   VAR_IN_OUT
      iqUDT_FifoRcvHeader : "UDT_FifoHeader";   // FIFO receive header
      iqs_FifoRcvData : Array[*] of "UDT_Message";   // FIFO receive data
      iqUDT_FifoMedPriorityHLC : "UDT_FifoHeader";   // FIFO UDS send Header
      iqa_FifoMedPriorityHLC : Array[*] of "UDT_Message";   // FIFO UDS send data
      iqUDT_HLCCommands : "UDT_FedExCommands";   // Commands from UDS
      iqUDT_DA : Struct   // Destination assignment message
         NewMessage : Bool;   // New message received from UDS
         Data : "UDT_FedExMessageDaRa";   // Destination assignment message body
      END_STRUCT;
      iqUDT_RA : Struct   // Destination re-assignment message
         NewMessage : Bool;   // New message received from UDS
         Data : "UDT_FedExMessageDaRa";   // Destination re-assignment message body
      END_STRUCT;
      iqUDT_CD : Struct   // Command message
         NewMessage : Bool;   // New message received from UDS
         Data : "UDT_FedExMessageCD";   // Command message body
      END_STRUCT;
      iqUDT_PS : Struct   // Parameters set message
         NewMessage : Bool;   // New message received from UDS
         Data : "UDT_FedExMessagePS";   // Parameters set message body
      END_STRUCT;
      iqUDT_CustomerIDReference : "UDT_FedExCustomerID";
      iqx_SendHB { ExternalAccessible := 'False'; ExternalVisible := 'False'; ExternalWritable := 'False'} : Bool;   // Send heartbeat request
      iqx_ResetListeningTimer { ExternalAccessible := 'False'; ExternalVisible := 'False'; ExternalWritable := 'False'} : Bool;   // Reset listening time in Heartbeat block
      iq_LoginOK { ExternalAccessible := 'False'; ExternalVisible := 'False'; ExternalWritable := 'False'} : Bool;   // Login in UDS ok
   END_VAR

   VAR
      sFB_FedExLoginResponse { ExternalAccessible := 'False'; ExternalVisible := 'False'; ExternalWritable := 'False'; S7_SetPoint := 'False'} : "FB_FedExLoginResponse";   // Login request send
      sUDT_Facillity { ExternalAccessible := 'False'; ExternalVisible := 'False'; ExternalWritable := 'False'; S7_SetPoint := 'False'} : "UDT_FedExFacility";   // System configuration
      sUDT_MSGHeader { ExternalAccessible := 'False'; ExternalVisible := 'False'; ExternalWritable := 'False'; S7_SetPoint := 'False'} : "UDT_FedExMessageHeader";   // Message header
      sUDT_FifoMsg { ExternalAccessible := 'False'; ExternalVisible := 'False'; ExternalWritable := 'False'; S7_SetPoint := 'False'} : "UDT_Message";   // Buffer for fifos message
      sa_Status { ExternalAccessible := 'False'; ExternalVisible := 'False'; ExternalWritable := 'False'} : Struct   // Status structure
         FIFORcvStatus { ExternalAccessible := 'False'; ExternalVisible := 'False'; ExternalWritable := 'False'} : "UDT_FifoStatus";   // Receive FIFO status structure
         FIFOError { ExternalAccessible := 'False'; ExternalVisible := 'False'; ExternalWritable := 'False'; S7_SetPoint := 'True'} : Bool;   // FIFO error
         FIFOWarning { ExternalAccessible := 'False'; ExternalVisible := 'False'; ExternalWritable := 'False'; S7_SetPoint := 'True'} : Bool;   // FIFO warning
         InvalidCommandCode { ExternalAccessible := 'False'; ExternalVisible := 'False'; ExternalWritable := 'False'} : Bool;   // Invalid command code
         InvalidType { ExternalAccessible := 'False'; ExternalVisible := 'False'; ExternalWritable := 'False'; S7_SetPoint := 'True'} : Bool;   // Invalid message type
         InvalidParameterID { ExternalAccessible := 'False'; ExternalVisible := 'False'; ExternalWritable := 'False'} : Bool;   // Invalig parameter ID
         InvalidLength { ExternalAccessible := 'False'; ExternalVisible := 'False'; ExternalWritable := 'False'} : Bool;   // Received message length is different than programmed
      END_STRUCT;
      st_TimeToSet {InstructionName := 'DTL'; LibVersion := '1.0'; ExternalAccessible := 'False'; ExternalVisible := 'False'; ExternalWritable := 'False'} : DTL;   // Time received from HLC used to set time in the PLC
      ss_NNNNNN { ExternalAccessible := 'False'; ExternalVisible := 'False'; ExternalWritable := 'False'} : String[6];   // GIN number extracted from Package ID
      ss_SS { ExternalAccessible := 'False'; ExternalVisible := 'False'; ExternalWritable := 'False'} : String[2];   // Maximum frequency of the messages
      ss_SorterNumber { ExternalAccessible := 'False'; ExternalVisible := 'False'; ExternalWritable := 'False'} : String;   // Sorter number
      ss_DiverterNumber { ExternalAccessible := 'False'; ExternalVisible := 'False'; ExternalWritable := 'False'} : String;   // Diverter number
      si_GIN { ExternalAccessible := 'False'; ExternalVisible := 'False'; ExternalWritable := 'False'} : Int;   // Gin number converted from string to int
      si_ChuteNumber { ExternalAccessible := 'False'; ExternalVisible := 'False'; ExternalWritable := 'False'} : Int;   // Chute number to enable/disable purge
      si_SS { ExternalAccessible := 'False'; ExternalVisible := 'False'; ExternalWritable := 'False'} : Int;   // Maximum frequency of the messages
      si_i { ExternalAccessible := 'False'; ExternalVisible := 'False'; ExternalWritable := 'False'} : Int;   // Loop counter
      si_PositionOfSpace { ExternalAccessible := 'False'; ExternalVisible := 'False'; ExternalWritable := 'False'} : Int;   // Position of spaces used to remove spaces
      si_MessageLegth { ExternalAccessible := 'False'; ExternalVisible := 'False'; ExternalWritable := 'False'} : Int;   // Received message length
      si_ComValueLen { ExternalAccessible := 'False'; ExternalVisible := 'False'; ExternalWritable := 'False'} : Int;   // Command value length
      si_SpacePositionComValue { ExternalAccessible := 'False'; ExternalVisible := 'False'; ExternalWritable := 'False'} : Int;   // Position of spaces used to remove spaces
      si_WriteTimeStatus { ExternalAccessible := 'False'; ExternalVisible := 'False'; ExternalWritable := 'False'} : Int;   // WR_LOC_T Status
      si_CustomerID { ExternalAccessible := 'False'; ExternalVisible := 'False'; ExternalWritable := 'False'} : Int;
      sx_FacialityCheck { ExternalAccessible := 'False'; ExternalVisible := 'False'; ExternalWritable := 'False'} : Bool;   // When TRUE received faciality configuration is the same as configured in the PLC
      sx_LogOffRequest { ExternalAccessible := 'False'; ExternalVisible := 'False'; ExternalWritable := 'False'} : Bool;   // Log off request from UDS
   END_VAR

   VAR_TEMP
      tx_MsgRead : Bool;   // Message read from FIFO
   END_VAR

   VAR CONSTANT
      cs_DA : String := 'DA';   // Destination assignment message type
      cs_RA : String := 'RA';   // Destination re-assignment message type
      cs_HB : String := 'HB';   // Heartbeat message type
      cs_LI : String := 'LI';   // Login request message type
      cs_LS : String := 'LS';   // Log-off message type
      cs_CD : String := 'CD';   // Command message type
      cs_PS : String := 'PS';   // Parameter set message type
      ci_SizeDAMessage : Int := 213;   // Destination assignment message length
      ci_SizeRAMessage : Int := 213;   // Destination re-assignment message length
      ci_SizeLIMessage : Int := 35;   // Login request message length
      ci_SizeCDMessage : Int := 113;   // Command message length
      ci_SizePSMessage : Int := 129;   // Parameter set message length
   END_VAR


BEGIN
	(*
	----------------------------------------------------------------------------------------

	Version history:
	Date        | Version   | Author        | Remark
	----------------------------------------------------------------------------------------
	22/07/2021  | 1.0       | J.Krawczuk    | first release MHS TIA 15.1
	11/04/2022  | 1.1       | K.Pokorski    | Review
	21/02/2023  | 4.0       | F.Baten       | 4.0 Release TIA 17.5
	*)

	REGION 1 – FIFO header status update

	    // Mode 'S' - FIFO register status update
	    "FC_Fifo"(ic_Mode := 'S',
	              qUDT_Status => #sa_Status.FIFORcvStatus,
	              qx_Error => #sa_Status.FIFOError,
	              qx_Warning => #sa_Status.FIFOWarning,
	              iqv_Data := #sUDT_FifoMsg,
	              iqUDT_FifoHeader := #iqUDT_FifoRcvHeader,
	              iqv_DataBuffer := #iqs_FifoRcvData);

	    IF (NOT #iqUDT_FifoRcvHeader.Status.Empty                             // FIFO not empty
	        AND NOT #sa_Status.FIFOError)                                      // No FIFO error
	    THEN

	        // Mode 'R' - Read FIFO record
	        "FC_Fifo"(ic_Mode := 'R',
	                  qUDT_Status => #sa_Status.FIFORcvStatus,
	                  qx_Error => #sa_Status.FIFOError,
	                  qx_Warning => #sa_Status.FIFOWarning,
	                  iqv_Data := #sUDT_FifoMsg,
	                  iqUDT_FifoHeader := #iqUDT_FifoRcvHeader,
	                  iqv_DataBuffer := #iqs_FifoRcvData);

	        // Message read bit set and position initialize
	        #tx_MsgRead := TRUE;

	        // FIFO empty or FIFO error occured
	    ELSE

	        #tx_MsgRead := FALSE;

	    END_IF;

	END_REGION

	REGION 2 – Decoding header

	    IF #tx_MsgRead      // New message
	    THEN
	        // Header decode
	        "FC_FedExDecodeHeader"(iUDT_FifoMsg := #sUDT_FifoMsg,
	                               qUDT_MSGHeader => #sUDT_MSGHeader);
	    END_IF;
	END_REGION

	REGION 3 - Decoding body

	    IF #tx_MsgRead                                                              // New message
	    THEN
	        #si_MessageLegth := STRING_TO_INT(#sUDT_MSGHeader.MessageLength);      // Convert message length to integer
	        #sa_Status.InvalidType := FALSE;                                        // Invalid type status initialize

	        // Login request message
	        IF #sUDT_MSGHeader.MessageType = #cs_LI
	        THEN

	            // Received message length validation
	            IF #si_MessageLegth = #ci_SizeLIMessage
	            THEN

	                // Faciality ID
	                Chars_TO_Strg(Chars := #sUDT_FifoMsg.Character,
	                              pChars := 7,
	                              Cnt := 6,
	                              Strg => #sUDT_Facillity.FacilityID);

	                // System ID
	                Chars_TO_Strg(Chars := #sUDT_FifoMsg.Character,
	                              pChars := 13,
	                              Cnt := 15,
	                              Strg => #sUDT_Facillity.SystemID);

	                // Version ID
	                Chars_TO_Strg(Chars := #sUDT_FifoMsg.Character,
	                              pChars := 28,
	                              Cnt := 6,
	                              Strg => #sUDT_Facillity.VersionID);

	                // Maximum message frequency
	                Chars_TO_Strg(Chars := #sUDT_FifoMsg.Character,
	                              pChars := 34,
	                              Cnt := 2,
	                              Strg => #ss_SS);

	                // Maximum message frequency conversion to integer
	                #si_SS := STRING_TO_INT(#ss_SS);

	                // For loop to remove spaces from Version ID
	                FOR #si_i := 1 TO 6 DO

	                    #si_PositionOfSpace := 0;
	                    #si_PositionOfSpace := FIND(IN1 := #sUDT_Facillity.VersionID, IN2 := ' ');

	                    IF #si_PositionOfSpace > 0
	                    THEN
	                        #sUDT_Facillity.VersionID := DELETE(IN := #sUDT_Facillity.VersionID, L := 1, P := #si_PositionOfSpace);

	                    END_IF;

	                END_FOR;

	                // Checking if received facility configuration matches configuration in the PLC
	                #sx_FacialityCheck := #iUDT_FacilitySystem.FacilityID = #sUDT_Facillity.FacilityID
	                AND #iUDT_FacilitySystem.SystemID = #sUDT_Facillity.SystemID
	                AND #iUDT_FacilitySystem.VersionID = #sUDT_Facillity.VersionID
	                AND #iUDT_FacilitySystem.SS = #si_SS;

	                // Login response message send
	                #sFB_FedExLoginResponse(iUDT_Facility := #iUDT_FacilityPLC,
	                                        is_LastHost := #is_LastHost,
	                                        ix_ConnectionStatus := #sx_FacialityCheck,
	                                        iqUDT_FifoHeader := #iqUDT_FifoMedPriorityHLC,
	                                        iqa_FifoData := #iqa_FifoMedPriorityHLC);

	                #iqx_ResetListeningTimer := TRUE;
	                #iq_LoginOK := #sx_FacialityCheck;
	            ELSE

	                // In case when received message length is different than programmed set error
	                #sa_Status.InvalidLength := TRUE;

	            END_IF;

	            // Log-off request message
	        ELSIF #sUDT_MSGHeader.MessageType = #cs_LS
	        THEN
	            #sx_LogOffRequest := TRUE;

	            // Destination assignment message
	        ELSIF #sUDT_MSGHeader.MessageType = #cs_DA
	        THEN

	            // Received message length validation
	            IF #si_MessageLegth = #ci_SizeDAMessage
	            THEN

	                // LLC system ID
	                Chars_TO_Strg(Chars := #sUDT_FifoMsg.Character,
	                              pChars := 7,
	                              Cnt := 15,
	                              Strg => #iqUDT_DA.Data.LLCSystemID);

	                // Package ID
	                Chars_TO_Strg(Chars := #sUDT_FifoMsg.Character,
	                              pChars := 22,
	                              Cnt := 15,
	                              Strg => #iqUDT_DA.Data.PackageID);

	                // High level package ID
	                Chars_TO_Strg(Chars := #sUDT_FifoMsg.Character,
	                              pChars := 37,
	                              Cnt := 10,
	                              Strg => #iqUDT_DA.Data.HLCPackageID);

	                // Cell number
	                Chars_TO_Strg(Chars := #sUDT_FifoMsg.Character,
	                              pChars := 47,
	                              Cnt := 4,
	                              Strg => #iqUDT_DA.Data.CellNumber);

	                // Destination 1
	                Chars_TO_Strg(Chars := #sUDT_FifoMsg.Character,
	                              pChars := 51,
	                              Cnt := 6,
	                              Strg => #iqUDT_DA.Data.Destination1);

	                // Cut off time destination 1
	                Chars_TO_Strg(Chars := #sUDT_FifoMsg.Character,
	                              pChars := 57,
	                              Cnt := 5,
	                              Strg => #iqUDT_DA.Data.CutOffTimeDestination1);

	                // Destination 2
	                Chars_TO_Strg(Chars := #sUDT_FifoMsg.Character,
	                              pChars := 62,
	                              Cnt := 6,
	                              Strg => #iqUDT_DA.Data.Destination2);

	                // Cut off time destination 2
	                Chars_TO_Strg(Chars := #sUDT_FifoMsg.Character,
	                              pChars := 68,
	                              Cnt := 5,
	                              Strg => #iqUDT_DA.Data.CutOffTimeDestination2);

	                // Destination 3
	                Chars_TO_Strg(Chars := #sUDT_FifoMsg.Character,
	                              pChars := 73,
	                              Cnt := 6,
	                              Strg => #iqUDT_DA.Data.Destination3);

	                // Cut off time destination 3
	                Chars_TO_Strg(Chars := #sUDT_FifoMsg.Character,
	                              pChars := 79,
	                              Cnt := 5,
	                              Strg => #iqUDT_DA.Data.CutOffTimeDestination3);

	                // Destination 4
	                Chars_TO_Strg(Chars := #sUDT_FifoMsg.Character,
	                              pChars := 84,
	                              Cnt := 6,
	                              Strg => #iqUDT_DA.Data.Destination4);

	                // Cut off time destination 4
	                Chars_TO_Strg(Chars := #sUDT_FifoMsg.Character,
	                              pChars := 90,
	                              Cnt := 5,
	                              Strg => #iqUDT_DA.Data.CutOffTimeDestination4);

	                // Destination 5
	                Chars_TO_Strg(Chars := #sUDT_FifoMsg.Character,
	                              pChars := 95,
	                              Cnt := 6,
	                              Strg => #iqUDT_DA.Data.Destination5);

	                // Cut off time destination 5
	                Chars_TO_Strg(Chars := #sUDT_FifoMsg.Character,
	                              pChars := 101,
	                              Cnt := 5,
	                              Strg => #iqUDT_DA.Data.CutOffTimeDestination5);

	                // High level data text
	                Chars_TO_Strg(Chars := #sUDT_FifoMsg.Character,
	                              pChars := 106,
	                              Cnt := 20,
	                              Strg => #iqUDT_DA.Data.HLCDataText);

	                // Barcode data
	                Chars_TO_Strg(Chars := #sUDT_FifoMsg.Character,
	                              pChars := 126,
	                              Cnt := 50,
	                              Strg => #iqUDT_DA.Data.Barcodedata);

	                // Result code
	                Chars_TO_Strg(Chars := #sUDT_FifoMsg.Character,
	                              pChars := 176,
	                              Cnt := 16,
	                              Strg => #iqUDT_DA.Data.HLCResultCode);

	                // Timestamp
	                Chars_TO_Strg(Chars := #sUDT_FifoMsg.Character,
	                              pChars := 192,
	                              Cnt := 17,
	                              Strg => #iqUDT_DA.Data.Timestamp);

	                // Time zone designator
	                Chars_TO_Strg(Chars := #sUDT_FifoMsg.Character,
	                              pChars := 209,
	                              Cnt := 5,
	                              Strg => #iqUDT_DA.Data.TimeZoneDesignator);

	                // Convert 'NNNNNN' part in package ID to GIN number and store data in GIN database
	                #ss_NNNNNN := RIGHT(IN := #iqUDT_DA.Data.PackageID, L := 6);
	                STRG_VAL(IN := #ss_NNNNNN,
	                         FORMAT := 16#0,
	                         P := 1,
	                         OUT => #si_CustomerID);

	                IF #si_CustomerID > 1 AND #si_CustomerID < 999999 THEN
	                    #si_GIN := #iqUDT_CustomerIDReference.CustomerIDReference[#si_CustomerID];
	                END_IF;

	                // Write data from destination assignment message to GIN array
	                IF #si_GIN > 0
	                    AND #si_GIN <= 9999
	                THEN

	                    "DB_GIN".GIN[#si_GIN].FedEx.LLCSystemID := #iqUDT_DA.Data.LLCSystemID;
	                    "DB_GIN".GIN[#si_GIN].FedEx.PackageID := #iqUDT_DA.Data.PackageID;
	                    "DB_GIN".GIN[#si_GIN].FedEx.HLCPackageID := #iqUDT_DA.Data.HLCPackageID;
	                    "DB_GIN".GIN[#si_GIN].FedEx.CellNumber := #iqUDT_DA.Data.CellNumber;
	                    "DB_GIN".GIN[#si_GIN].FedEx.Destination1 := #iqUDT_DA.Data.Destination1;
	                    "DB_GIN".GIN[#si_GIN].FedEx.CutOffTimeDestination1 := #iqUDT_DA.Data.CutOffTimeDestination1;
	                    "DB_GIN".GIN[#si_GIN].FedEx.Destination2 := #iqUDT_DA.Data.Destination2;
	                    "DB_GIN".GIN[#si_GIN].FedEx.CutOffTimeDestination2 := #iqUDT_DA.Data.CutOffTimeDestination2;
	                    "DB_GIN".GIN[#si_GIN].FedEx.Destination3 := #iqUDT_DA.Data.Destination3;
	                    "DB_GIN".GIN[#si_GIN].FedEx.CutOffTimeDestination3 := #iqUDT_DA.Data.CutOffTimeDestination3;
	                    "DB_GIN".GIN[#si_GIN].FedEx.Destination4 := #iqUDT_DA.Data.Destination4;
	                    "DB_GIN".GIN[#si_GIN].FedEx.CutOffTimeDestination4 := #iqUDT_DA.Data.CutOffTimeDestination4;
	                    "DB_GIN".GIN[#si_GIN].FedEx.Destination5 := #iqUDT_DA.Data.Destination5;
	                    "DB_GIN".GIN[#si_GIN].FedEx.CutOffTimeDestination5 := #iqUDT_DA.Data.CutOffTimeDestination5;
	                    "DB_GIN".GIN[#si_GIN].FedEx.HLCDataText := #iqUDT_DA.Data.HLCDataText;
	                    "DB_GIN".GIN[#si_GIN].FedEx.Barcodedata := #iqUDT_DA.Data.Barcodedata;
	                    "DB_GIN".GIN[#si_GIN].FedEx.HLCResultCode := #iqUDT_DA.Data.HLCResultCode;
	                    "DB_GIN".GIN[#si_GIN].FedEx.Timestamp := #iqUDT_DA.Data.Timestamp;
	                    "DB_GIN".GIN[#si_GIN].FedEx.TimeZoneDesignator := #iqUDT_DA.Data.TimeZoneDesignator;

	                    "DB_GIN".GIN[#si_GIN].General.Destination[0] := STRING_TO_DINT(#iqUDT_DA.Data.Destination1);
	                    "DB_GIN".GIN[#si_GIN].General.Destination[1] := STRING_TO_DINT(#iqUDT_DA.Data.Destination2);
	                    "DB_GIN".GIN[#si_GIN].General.Destination[2] := STRING_TO_DINT(#iqUDT_DA.Data.Destination3);
	                    "DB_GIN".GIN[#si_GIN].General.Destination[3] := STRING_TO_DINT(#iqUDT_DA.Data.Destination4);
	                    "DB_GIN".GIN[#si_GIN].General.Destination[4] := STRING_TO_DINT(#iqUDT_DA.Data.Destination5);

	                    #iqUDT_DA.NewMessage := TRUE;
	                    #iqx_ResetListeningTimer := TRUE;

	                END_IF;
	            ELSE
	                // In case when received message length is different than programmed set error
	                #sa_Status.InvalidLength := TRUE;

	            END_IF;

	            // Destination re-assignment message
	        ELSIF #sUDT_MSGHeader.MessageType = #cs_RA
	        THEN

	            // Received message length validation
	            IF #si_MessageLegth = #ci_SizeRAMessage
	            THEN

	                // LLC system ID
	                Chars_TO_Strg(Chars := #sUDT_FifoMsg.Character,
	                              pChars := 7,
	                              Cnt := 15,
	                              Strg => #iqUDT_RA.Data.LLCSystemID);

	                // Package ID
	                Chars_TO_Strg(Chars := #sUDT_FifoMsg.Character,
	                              pChars := 22,
	                              Cnt := 15,
	                              Strg => #iqUDT_RA.Data.PackageID);

	                // High level package ID
	                Chars_TO_Strg(Chars := #sUDT_FifoMsg.Character,
	                              pChars := 37,
	                              Cnt := 10,
	                              Strg => #iqUDT_RA.Data.HLCPackageID);

	                // Cell number
	                Chars_TO_Strg(Chars := #sUDT_FifoMsg.Character,
	                              pChars := 47,
	                              Cnt := 4,
	                              Strg => #iqUDT_RA.Data.CellNumber);

	                // Destination 1
	                Chars_TO_Strg(Chars := #sUDT_FifoMsg.Character,
	                              pChars := 51,
	                              Cnt := 6,
	                              Strg => #iqUDT_RA.Data.Destination1);

	                // Cut off time destination 1
	                Chars_TO_Strg(Chars := #sUDT_FifoMsg.Character,
	                              pChars := 57,
	                              Cnt := 5,
	                              Strg => #iqUDT_RA.Data.CutOffTimeDestination1);

	                // Destination 2
	                Chars_TO_Strg(Chars := #sUDT_FifoMsg.Character,
	                              pChars := 62,
	                              Cnt := 6,
	                              Strg => #iqUDT_RA.Data.Destination2);

	                // Cut off time destination 2
	                Chars_TO_Strg(Chars := #sUDT_FifoMsg.Character,
	                              pChars := 68,
	                              Cnt := 5,
	                              Strg => #iqUDT_RA.Data.CutOffTimeDestination2);

	                // Destination 3
	                Chars_TO_Strg(Chars := #sUDT_FifoMsg.Character,
	                              pChars := 73,
	                              Cnt := 6,
	                              Strg => #iqUDT_RA.Data.Destination3);

	                // Cut off time destination 3
	                Chars_TO_Strg(Chars := #sUDT_FifoMsg.Character,
	                              pChars := 79,
	                              Cnt := 5,
	                              Strg => #iqUDT_RA.Data.CutOffTimeDestination3);

	                // Destination 4
	                Chars_TO_Strg(Chars := #sUDT_FifoMsg.Character,
	                              pChars := 84,
	                              Cnt := 6,
	                              Strg => #iqUDT_RA.Data.Destination4);

	                // Cut off time destination 4
	                Chars_TO_Strg(Chars := #sUDT_FifoMsg.Character,
	                              pChars := 90,
	                              Cnt := 5,
	                              Strg => #iqUDT_RA.Data.CutOffTimeDestination4);

	                // Destination 5
	                Chars_TO_Strg(Chars := #sUDT_FifoMsg.Character,
	                              pChars := 95,
	                              Cnt := 6,
	                              Strg => #iqUDT_RA.Data.Destination5);

	                // Cut off time destination 5
	                Chars_TO_Strg(Chars := #sUDT_FifoMsg.Character,
	                              pChars := 101,
	                              Cnt := 5,
	                              Strg => #iqUDT_RA.Data.CutOffTimeDestination5);

	                // High level data text
	                Chars_TO_Strg(Chars := #sUDT_FifoMsg.Character,
	                              pChars := 106,
	                              Cnt := 20,
	                              Strg => #iqUDT_RA.Data.HLCDataText);

	                // Barcode data
	                Chars_TO_Strg(Chars := #sUDT_FifoMsg.Character,
	                              pChars := 126,
	                              Cnt := 50,
	                              Strg => #iqUDT_RA.Data.Barcodedata);

	                // Result code
	                Chars_TO_Strg(Chars := #sUDT_FifoMsg.Character,
	                              pChars := 176,
	                              Cnt := 16,
	                              Strg => #iqUDT_RA.Data.HLCResultCode);

	                // Timestamp
	                Chars_TO_Strg(Chars := #sUDT_FifoMsg.Character,
	                              pChars := 192,
	                              Cnt := 17,
	                              Strg => #iqUDT_RA.Data.Timestamp);

	                // Time zone designator
	                Chars_TO_Strg(Chars := #sUDT_FifoMsg.Character,
	                              pChars := 209,
	                              Cnt := 5,
	                              Strg => #iqUDT_RA.Data.TimeZoneDesignator);

	                // Convert 'NNNNNN' part in package ID to GIN number and store data in GIN database
	                #ss_NNNNNN := RIGHT(IN := #iqUDT_RA.Data.PackageID, L := 6);
	                STRG_VAL(IN := #ss_NNNNNN,
	                         FORMAT := 16#0,
	                         P := 1,
	                         OUT => #si_CustomerID);

	                IF #si_CustomerID > 1 AND #si_CustomerID < 999999 THEN
	                    #si_GIN := #iqUDT_CustomerIDReference.CustomerIDReference[#si_CustomerID];
	                END_IF;

	                // Write data from destination assignment message to GIN array
	                IF #si_GIN > 0
	                    AND #si_GIN <= 9999
	                THEN
	                    "DB_GIN".GIN[#si_GIN].FedEx.LLCSystemID := #iqUDT_RA.Data.LLCSystemID;
	                    "DB_GIN".GIN[#si_GIN].FedEx.PackageID := #iqUDT_RA.Data.PackageID;
	                    "DB_GIN".GIN[#si_GIN].FedEx.HLCPackageID := #iqUDT_RA.Data.HLCPackageID;
	                    "DB_GIN".GIN[#si_GIN].FedEx.CellNumber := #iqUDT_RA.Data.CellNumber;
	                    "DB_GIN".GIN[#si_GIN].FedEx.Destination1 := #iqUDT_RA.Data.Destination1;
	                    "DB_GIN".GIN[#si_GIN].FedEx.CutOffTimeDestination1 := #iqUDT_RA.Data.CutOffTimeDestination1;
	                    "DB_GIN".GIN[#si_GIN].FedEx.Destination2 := #iqUDT_RA.Data.Destination2;
	                    "DB_GIN".GIN[#si_GIN].FedEx.CutOffTimeDestination2 := #iqUDT_RA.Data.CutOffTimeDestination2;
	                    "DB_GIN".GIN[#si_GIN].FedEx.Destination3 := #iqUDT_RA.Data.Destination3;
	                    "DB_GIN".GIN[#si_GIN].FedEx.CutOffTimeDestination3 := #iqUDT_RA.Data.CutOffTimeDestination3;
	                    "DB_GIN".GIN[#si_GIN].FedEx.Destination4 := #iqUDT_RA.Data.Destination4;
	                    "DB_GIN".GIN[#si_GIN].FedEx.CutOffTimeDestination4 := #iqUDT_RA.Data.CutOffTimeDestination4;
	                    "DB_GIN".GIN[#si_GIN].FedEx.Destination5 := #iqUDT_RA.Data.Destination5;
	                    "DB_GIN".GIN[#si_GIN].FedEx.CutOffTimeDestination5 := #iqUDT_RA.Data.CutOffTimeDestination5;
	                    "DB_GIN".GIN[#si_GIN].FedEx.HLCDataText := #iqUDT_RA.Data.HLCDataText;
	                    "DB_GIN".GIN[#si_GIN].FedEx.Barcodedata := #iqUDT_RA.Data.Barcodedata;
	                    "DB_GIN".GIN[#si_GIN].FedEx.HLCResultCode := #iqUDT_RA.Data.HLCResultCode;
	                    "DB_GIN".GIN[#si_GIN].FedEx.Timestamp := #iqUDT_RA.Data.Timestamp;
	                    "DB_GIN".GIN[#si_GIN].FedEx.TimeZoneDesignator := #iqUDT_RA.Data.TimeZoneDesignator;

	                    "DB_GIN".GIN[#si_GIN].General.Destination[0] := STRING_TO_DINT(#iqUDT_RA.Data.Destination1);
	                    "DB_GIN".GIN[#si_GIN].General.Destination[1] := STRING_TO_DINT(#iqUDT_RA.Data.Destination2);
	                    "DB_GIN".GIN[#si_GIN].General.Destination[2] := STRING_TO_DINT(#iqUDT_RA.Data.Destination3);
	                    "DB_GIN".GIN[#si_GIN].General.Destination[3] := STRING_TO_DINT(#iqUDT_RA.Data.Destination4);
	                    "DB_GIN".GIN[#si_GIN].General.Destination[4] := STRING_TO_DINT(#iqUDT_RA.Data.Destination5);

	                    #iqUDT_RA.NewMessage := TRUE;
	                    #iqx_ResetListeningTimer := TRUE;

	                END_IF;

	            ELSE
	                // In case when received message length is different than programmed set error
	                #sa_Status.InvalidLength := TRUE;

	            END_IF;

	            // Command message
	        ELSIF #sUDT_MSGHeader.MessageType = #cs_CD
	        THEN
	            // Received message length validation
	            IF #si_MessageLegth = #ci_SizeCDMessage
	            THEN
	                // Invalid command code initialization
	                #sa_Status.InvalidCommandCode := FALSE;

	                // Command code
	                Chars_TO_Strg(Chars := #sUDT_FifoMsg.Character,
	                              pChars := 7,
	                              Cnt := 3,
	                              Strg => #iqUDT_CD.Data.CommandCode);

	                // Command value
	                Chars_TO_Strg(Chars := #sUDT_FifoMsg.Character,
	                              pChars := 10,
	                              Cnt := 82,
	                              Strg => #iqUDT_CD.Data.CommandValue);

	                // Timestamp
	                Chars_TO_Strg(Chars := #sUDT_FifoMsg.Character,
	                              pChars := 92,
	                              Cnt := 17,
	                              Strg => #iqUDT_CD.Data.Timestamp);

	                // Time zone designator
	                Chars_TO_Strg(Chars := #sUDT_FifoMsg.Character,
	                              pChars := 109,
	                              Cnt := 5,
	                              Strg => #iqUDT_CD.Data.TimeZoneDesignator);

	                #iqUDT_CD.NewMessage := TRUE;
	                #iqx_ResetListeningTimer := TRUE;

	                // Start of sort command
	                IF #iqUDT_CD.Data.CommandCode = '001'
	                THEN
	                    #iqUDT_HLCCommands.StartSort.StartSort := TRUE;
	                    #iqUDT_HLCCommands.EndSort.EndSort := FALSE;
	                    #iqUDT_HLCCommands.StartSort.NewMessage := TRUE;

	                    // End of sort command
	                ELSIF #iqUDT_CD.Data.CommandCode = '002'
	                THEN
	                    #iqUDT_HLCCommands.StartSort.StartSort := FALSE;
	                    #iqUDT_HLCCommands.EndSort.EndSort := TRUE;
	                    #iqUDT_HLCCommands.EndSort.NewMessage := TRUE;
	                    // Upload chute status command
	                ELSIF #iqUDT_CD.Data.CommandCode = '003'
	                THEN
	                    #iqUDT_HLCCommands.UploadChuteStatus.NewMessage := TRUE;

	                    // Upload all equipment status command
	                ELSIF #iqUDT_CD.Data.CommandCode = '004'
	                THEN
	                    #iqUDT_HLCCommands.UploadAllStatus.NewMessage := TRUE;

	                    // Block diverter automated smalls
	                ELSIF #iqUDT_CD.Data.CommandCode = '005'
	                THEN
	                    #ss_SorterNumber := MID(IN := #iqUDT_CD.Data.CommandValue, L := 5, P := 3);
	                    #ss_DiverterNumber := MID(IN := #iqUDT_CD.Data.CommandValue, L := 6, P := 8);
	                    #iqUDT_HLCCommands.BlockDivertSmalls.SorterNumber := (#ss_SorterNumber);
	                    #iqUDT_HLCCommands.BlockDivertSmalls.DivertNumber := (#ss_DiverterNumber);

	                    // Unblock diverter automated smalls
	                ELSIF #iqUDT_CD.Data.CommandCode = '006'
	                THEN

	                    #ss_SorterNumber := MID(IN := #iqUDT_CD.Data.CommandValue, L := 5, P := 3);
	                    #ss_DiverterNumber := MID(IN := #iqUDT_CD.Data.CommandValue, L := 6, P := 8);
	                    #iqUDT_HLCCommands.UnblockDivertSmalls.SorterNumber := (#ss_SorterNumber);
	                    #iqUDT_HLCCommands.UnblockDivertSmalls.DivertNumber := (#ss_DiverterNumber);

	                    // Chute purge enable
	                ELSIF #iqUDT_CD.Data.CommandCode = '007'
	                THEN

	                    // Removing spaces from caommand value
	                    FOR #si_i := 1 TO 82 DO

	                        #si_SpacePositionComValue := FIND(IN1 := #iqUDT_CD.Data.CommandValue, IN2 := ' ');
	                        IF #si_SpacePositionComValue <> 0
	                        THEN
	                            #iqUDT_CD.Data.CommandValue := DELETE(IN := #iqUDT_CD.Data.CommandValue, L := 1, P := #si_SpacePositionComValue);

	                        END_IF;

	                    END_FOR;

	                    #iqUDT_HLCCommands.EnablePurge.PLC := LEFT(IN := #iqUDT_CD.Data.CommandValue, L := 6);
	                    #iqUDT_CD.Data.CommandValue := DELETE(IN := #iqUDT_CD.Data.CommandValue, L := 6, P := 1);
	                    #si_ComValueLen := LEN(#iqUDT_CD.Data.CommandValue);

	                    // Extracting up to 5 chute numbers to enable purge
	                    IF #si_ComValueLen MOD 6 = 0 AND #si_ComValueLen <= 30
	                    THEN

	                        #si_ChuteNumber := 0;

	                        FOR #si_i := (#si_ComValueLen / 6) TO 1 BY -1 DO

	                            #si_ChuteNumber += 1;

	                            #iqUDT_HLCCommands.EnablePurge.Chute[#si_ChuteNumber] := (LEFT(IN := #iqUDT_CD.Data.CommandValue, L := 6));
	                            #iqUDT_CD.Data.CommandValue := DELETE(IN := #iqUDT_CD.Data.CommandValue, L := 6, P := 1);

	                        END_FOR;

	                    END_IF;

	                    // Chute purge disable
	                ELSIF #iqUDT_CD.Data.CommandCode = '008'
	                THEN
	                    // Removing spaces from caommand value
	                    FOR #si_i := 1 TO 82 DO

	                        #si_SpacePositionComValue := FIND(IN1 := #iqUDT_CD.Data.CommandValue, IN2 := ' ');
	                        IF #si_SpacePositionComValue <> 0
	                        THEN
	                            #iqUDT_CD.Data.CommandValue := DELETE(IN := #iqUDT_CD.Data.CommandValue, L := 1, P := #si_SpacePositionComValue);

	                        END_IF;

	                    END_FOR;

	                    #iqUDT_HLCCommands.DisablePurge.PLC := LEFT(IN := #iqUDT_CD.Data.CommandValue, L := 6);
	                    #iqUDT_CD.Data.CommandValue := DELETE(IN := #iqUDT_CD.Data.CommandValue, L := 6, P := 1);
	                    #si_ComValueLen := LEN(#iqUDT_CD.Data.CommandValue);

	                    // Extracting up to 5 chute numbers to disable purge
	                    IF #si_ComValueLen MOD 6 = 0
	                    THEN

	                        #si_ChuteNumber := 0;

	                        FOR #si_i := (#si_ComValueLen / 6) - 1 TO 1 BY -1 DO

	                            #si_ChuteNumber += 1;

	                            #iqUDT_HLCCommands.DisablePurge.Chute[#si_ChuteNumber] := (LEFT(IN := #iqUDT_CD.Data.CommandValue, L := 6));
	                            #iqUDT_CD.Data.CommandValue := DELETE(IN := #iqUDT_CD.Data.CommandValue, L := 6, P := 1);

	                        END_FOR;

	                    END_IF;

	                    // Lamp control
	                ELSIF #iqUDT_CD.Data.CommandCode = '009'
	                THEN

	                    #iqUDT_HLCCommands.ChuteLamp.ChuteNumber := (LEFT(IN := #iqUDT_CD.Data.CommandValue, L := 6));
	                    #iqUDT_HLCCommands.ChuteLamp.Mode := (MID(IN := #iqUDT_CD.Data.CommandValue, L := 1, P := 7));
	                    #iqUDT_HLCCommands.ChuteLamp.Color := (MID(IN := #iqUDT_CD.Data.CommandValue, L := 9, P := 8));

	                ELSE
	                    // In case when received command is different than programmed set error
	                    #sa_Status.InvalidCommandCode := TRUE;

	                END_IF;

	                //    #q_UDT_HLCCommands := #s_UDT_HLCCommands;

	            ELSE
	                // In case when received message length is different than programmed set error
	                #sa_Status.InvalidLength := TRUE;

	            END_IF;

	            // Parameter set message
	        ELSIF #sUDT_MSGHeader.MessageType = #cs_PS
	        THEN

	            // Received message length validation
	            IF #si_MessageLegth = #ci_SizePSMessage
	            THEN

	                // System ID
	                Chars_TO_Strg(Chars := #sUDT_FifoMsg.Character,
	                              pChars := 7,
	                              Cnt := 15,
	                              Strg => #iqUDT_PS.Data.SystemID);

	                // Parameter ID
	                Chars_TO_Strg(Chars := #sUDT_FifoMsg.Character,
	                              pChars := 22,
	                              Cnt := 4,
	                              Strg => #iqUDT_PS.Data.ParameterID);

	                // Parameter value
	                Chars_TO_Strg(Chars := #sUDT_FifoMsg.Character,
	                              pChars := 26,
	                              Cnt := 82,
	                              Strg => #iqUDT_PS.Data.ParameterValue);

	                // Timestamp
	                Chars_TO_Strg(Chars := #sUDT_FifoMsg.Character,
	                              pChars := 108,
	                              Cnt := 17,
	                              Strg => #iqUDT_PS.Data.Timestamp);

	                // Time zone designator
	                Chars_TO_Strg(Chars := #sUDT_FifoMsg.Character,
	                              pChars := 125,
	                              Cnt := 5,
	                              Strg => #iqUDT_PS.Data.TimeZoneDesignator);

	                #iqUDT_PS.NewMessage := TRUE;
	                #iqx_ResetListeningTimer := TRUE;

	                // Set time parameter
	                IF #iqUDT_PS.Data.ParameterID = 'TIME'
	                THEN
	                    // Invalid parameter ID initialization
	                    #sa_Status.InvalidParameterID := FALSE;

	                    // Converting received date and time to DTL format
	                    #st_TimeToSet.YEAR := STRING_TO_UINT(LEFT(IN := #iqUDT_PS.Data.ParameterValue, L := 4));
	                    #st_TimeToSet.MONTH := STRING_TO_USINT(MID(IN := #iqUDT_PS.Data.ParameterValue, L := 2, P := 5));
	                    #st_TimeToSet.DAY := STRING_TO_USINT(MID(IN := #iqUDT_PS.Data.ParameterValue, L := 2, P := 7));
	                    #st_TimeToSet.HOUR := STRING_TO_USINT(MID(IN := #iqUDT_PS.Data.ParameterValue, L := 2, P := 9));
	                    #st_TimeToSet.MINUTE := STRING_TO_USINT(MID(IN := #iqUDT_PS.Data.ParameterValue, L := 2, P := 11));
	                    #st_TimeToSet.SECOND := STRING_TO_USINT(MID(IN := #iqUDT_PS.Data.ParameterValue, L := 2, P := 13));
	                    #st_TimeToSet.NANOSECOND := 0;

	                    // Set time in the PLC
	                    #si_WriteTimeStatus := WR_LOC_T(LOCTIME := #st_TimeToSet, DST := FALSE);

	                ELSE
	                    // In case when received parameter ID is different than programmed set error
	                    #sa_Status.InvalidParameterID := TRUE;

	                END_IF;

	            ELSE
	                // In case when received message length is different than programmed set error
	                #sa_Status.InvalidLength := TRUE;

	            END_IF;

	            // Heartbeat message
	        ELSIF #sUDT_MSGHeader.MessageType = #cs_HB
	        THEN

	            #iqx_SendHB := TRUE;


	        ELSE
	            // In case when received message type is different than programmed set error
	            #sa_Status.InvalidType := TRUE;

	        END_IF;
	    END_IF;

	END_REGION
END_FUNCTION_BLOCK

FUNCTION_BLOCK "FB_FedExDestinationLookupMessage"
TITLE = FB_Heartbeat
{ S7_Optimized_Access := 'TRUE' }
AUTHOR : MHSE
FAMILY : UPS_SpecificCommunication
VERSION : 3.0
// ATTRIBUTES
// AUTO_NUMBER = True
// BLOCK_NUMBER = 67
// END_ATTRIBUTES
//Function block to send and monitor the UPS heartbeat message.
   VAR_INPUT
      iUDT_Facility { ExternalAccessible := 'False'; ExternalVisible := 'False'; ExternalWritable := 'False'} : "UDT_FedExFacility";   // System configuration
      is_LOConEquipment { ExternalAccessible := 'False'; ExternalVisible := 'False'; ExternalWritable := 'False'} : String[3];   // Location of the equipment
      is_DEPCOD { ExternalAccessible := 'False'; ExternalVisible := 'False'; ExternalWritable := 'False'} : String[6];   // Depot Code
      is_TYPofEquipment { ExternalAccessible := 'False'; ExternalVisible := 'False'; ExternalWritable := 'False'} : String[3];   // Type of equipment
      is_NumberOfTheEquipment { ExternalAccessible := 'False'; ExternalVisible := 'False'; ExternalWritable := 'False'} : String[3];   // Number of the equipment 001-999
      is_TrayCellNumber { ExternalAccessible := 'False'; ExternalVisible := 'False'; ExternalWritable := 'False'} : String[3];   // Tray/Cell number (for loop sorters) or generated by LLC (on line sorters).
      is_SorterNumber { ExternalAccessible := 'False'; ExternalVisible := 'False'; ExternalWritable := 'False'} : String[2];   // Sorter number
      is_InductionNumber { ExternalAccessible := 'False'; ExternalVisible := 'False'; ExternalWritable := 'False'} : String[2];   // Induction number
      is_AreaNumber { ExternalAccessible := 'False'; ExternalVisible := 'False'; ExternalWritable := 'False'} : String[2];   // Area number
      ii_Gin { ExternalAccessible := 'False'; ExternalVisible := 'False'; ExternalWritable := 'False'} : Int;   // GIN number
   END_VAR

   VAR_OUTPUT
      qx_Error { ExternalAccessible := 'False'; ExternalVisible := 'False'; ExternalWritable := 'False'} : Bool;   // Error
   END_VAR

   VAR_IN_OUT
      iqUDT_FifoHeader : "UDT_FifoHeader";   // FIFO header
      iqa_FifoData : Array[*] of "UDT_Message";   // FIFO data
      iqx_UnexpectedDLReq { ExternalAccessible := 'False'; ExternalVisible := 'False'; ExternalWritable := 'False'} : Bool;
   END_VAR

   VAR
      sUDT_MessageArray { ExternalAccessible := 'False'; ExternalVisible := 'False'; ExternalWritable := 'False'; S7_SetPoint := 'False'} : "UDT_Message";   // Message character array
      sa_Status { ExternalAccessible := 'False'; ExternalVisible := 'False'; ExternalWritable := 'False'} : Struct   // Status structure
         FIFOStatus { ExternalAccessible := 'False'; ExternalVisible := 'False'; ExternalWritable := 'False'} : "UDT_FifoStatus";   // FIFO status structure
         FIFOError { ExternalAccessible := 'False'; ExternalVisible := 'False'; ExternalWritable := 'False'; S7_SetPoint := 'True'} : Bool;   // FIFO data buffer full
         FIFOWarning { ExternalAccessible := 'False'; ExternalVisible := 'False'; ExternalWritable := 'False'; S7_SetPoint := 'True'} : Bool;   // FIFO error
         InvalidGIN { ExternalAccessible := 'False'; ExternalVisible := 'False'; ExternalWritable := 'False'} : Bool;   //  Invalid GIN
         InvalidMessageLength { ExternalAccessible := 'False'; ExternalVisible := 'False'; ExternalWritable := 'False'} : Bool;   // Calculated message length is different than required
         InvalidMsgArraySize { ExternalAccessible := 'False'; ExternalVisible := 'False'; ExternalWritable := 'False'} : Bool;   // Length of the message is bigger than length of message array
      END_STRUCT;
      sa_Statistics { ExternalAccessible := 'False'; ExternalVisible := 'False'; ExternalWritable := 'False'} : Struct   // Statistics structure
         NotSentWrongMsgLen { ExternalAccessible := 'False'; ExternalVisible := 'False'; ExternalWritable := 'False'} : DInt;   // COMISSIONING PURPOSE Messages not sent because built message length does not match with required message length
      END_STRUCT;
      ss_LLCSystemID { ExternalAccessible := 'False'; ExternalVisible := 'False'; ExternalWritable := 'False'} : String[15];   // Identifier of Low-Level controls
      ss_SequencialID { ExternalAccessible := 'False'; ExternalVisible := 'False'; ExternalWritable := 'False'} : String[6];   // Identifier of Low-Level controls
      ss_MessageP1 { ExternalAccessible := 'False'; ExternalVisible := 'False'; ExternalWritable := 'False'} : String;   // Message character string part 1
      ss_MessageP2 { ExternalAccessible := 'False'; ExternalVisible := 'False'; ExternalWritable := 'False'} : String;   // Message character string part 2
      ss_PackageID { ExternalAccessible := 'False'; ExternalVisible := 'False'; ExternalWritable := 'False'} : String[15];   // Identifier of Low-Level controls
      ss_Gap { ExternalAccessible := 'False'; ExternalVisible := 'False'; ExternalWritable := 'False'} : String[3];   // Gap converted to string
      sui_MsgArrayElNr { ExternalAccessible := 'False'; ExternalVisible := 'False'; ExternalWritable := 'False'} : UInt;   // Invalid message array size
      sui_ArrayOffset { ExternalAccessible := 'False'; ExternalVisible := 'False'; ExternalWritable := 'False'} : UInt;   // Offset for writing in the array
      si_OldGin { ExternalAccessible := 'False'; ExternalVisible := 'False'; ExternalWritable := 'False'} : Int;   // Previous Gin
      si_StringLen { ExternalAccessible := 'False'; ExternalVisible := 'False'; ExternalWritable := 'False'} : Int;   // Length of string used in loops to pad string with spaces or 0
      si_LenFillLoop { ExternalAccessible := 'False'; ExternalVisible := 'False'; ExternalWritable := 'False'} : Int;   // Loop couter
      si_MaxMsgLen { ExternalAccessible := 'False'; ExternalVisible := 'False'; ExternalWritable := 'False'} : Int;   // Maximum message length
      si_MsgLen { ExternalAccessible := 'False'; ExternalVisible := 'False'; ExternalWritable := 'False'} : Int;   // String character message length
      sx_Error { ExternalAccessible := 'False'; ExternalVisible := 'False'; ExternalWritable := 'False'} : Bool;
   END_VAR

   VAR CONSTANT
      cc_NULL : Char := '$00';   // NULL sign
      cc_STX : Char := '$02';   // Start of the text
      cc_ETX : Char := '$03';   // End of the text
      cs_Length : String := '0407';   // Legth of the message
      cs_MessageType : String := 'DL';   // Message type
   END_VAR


BEGIN
	(*
	----------------------------------------------------------------------------------------

	Version history:
	Date        | Version   | Author        | Remark
	----------------------------------------------------------------------------------------
	29/06/2021  | 1.0       | F.Baten       | first release MHS TIA 16.0
	04/08/2021  | 1.1       | J.Krawczuk    | Updating comments, changing message length
	10/11/2021  | 1.2       | M.Piela       | Updating regions numbering and interface changes
	05/04/2022  | 1.3       | K.Pokorski    | Review
	21/02/2023  | 4.0       | F.Baten       | 4.0 Release TIA 17.5
	*)

	REGION 1 – FIFO header status update

	    // Mode 'S' - FIFO register status update
	    "FC_Fifo"(ic_Mode := 'S',
	              qUDT_Status => #sa_Status.FIFOStatus,
	              qx_Error => #sa_Status.FIFOError,
	              qx_Warning => #sa_Status.FIFOWarning,
	              iqv_Data := #sUDT_MessageArray,
	              iqUDT_FifoHeader := #iqUDT_FifoHeader,
	              iqv_DataBuffer := #iqa_FifoData);
	END_REGION

	REGION 2 - GIN validation

	    // GIN validation
	    #sa_Status.InvalidGIN :=
	    #ii_Gin < 1
	    OR #ii_Gin > 9999;

	END_REGION

	REGION 3 – Message preparation
	    IF NOT #iqUDT_FifoHeader.Status.Full                       // FIFO isn't full
	        AND NOT #sa_Status.InvalidGIN
	        AND #ii_Gin <> #si_OldGin
	    THEN

	        REGION 3.1 - Sequential  ID
	            // ss_SequencialID character string clearing
	            #ss_SequencialID := '';
	            // ss_SequencialID integer input conversion to a character string
	            VAL_STRG(IN := "DB_GIN".GIN[#ii_Gin].FedEx.CustomerID,
	                     SIZE := 0,
	                     PREC := 0,
	                     FORMAT := 0,
	                     P := 1,
	                     OUT => #ss_SequencialID);
	            // Length of the ss_SequencialID character string
	            #si_StringLen := LEN(#ss_SequencialID);

	            // ss_SequencialID character string leading zeros addition
	            IF (#si_StringLen < 6)
	            THEN
	                FOR #si_LenFillLoop := 1 TO 6 - #si_StringLen DO
	                    #ss_SequencialID := CONCAT(IN1 := '0',
	                                               IN2 := #ss_SequencialID);
	                END_FOR;
	            END_IF;
	        END_REGION

	        REGION 3.2 LLC System ID
	            // Build LLC Syatem ID
	            #ss_LLCSystemID := CONCAT(IN1 := #is_DEPCOD,
	                                      IN2 := #is_LOConEquipment,
	                                      IN3 := #is_TYPofEquipment,
	                                      IN4 := #is_NumberOfTheEquipment);

	        END_REGION

	        REGION 3.3 - Package ID
	            // Build Package ID
	            #ss_PackageID := CONCAT(IN1 := #is_TrayCellNumber,
	                                    IN2 := #is_SorterNumber,
	                                    IN3 := #is_InductionNumber,
	                                    IN4 := #is_AreaNumber,
	                                    IN5 := #ss_SequencialID);
	        END_REGION

	        REGION 3.4 - Gap
	            // Gap character string clearing
	            #ss_Gap := '';

	            IF ("DB_GIN".GIN[#ii_Gin].General.LeadingGap > 999)
	            THEN
	                #ss_Gap := '999';
	            ELSE

	                // Gap integer input conversion to a character string
	                VAL_STRG(IN := "DB_GIN".GIN[#ii_Gin].General.LeadingGap,
	                         SIZE := 0,
	                         PREC := 0,
	                         FORMAT := 0,
	                         P := 1,
	                         OUT => #ss_Gap);
	                // Length of the gap character string
	                #si_StringLen := LEN(#ss_Gap);
	                // Gap character string leading zeros addition
	                IF (#si_StringLen < 3)
	                THEN
	                    FOR #si_LenFillLoop := 1 TO 3 - #si_StringLen DO
	                        #ss_Gap := CONCAT(IN1 := '0',
	                                          IN2 := #ss_Gap);
	                    END_FOR;

	                END_IF;

	            END_IF;


	        END_REGION

	        IF NOT #sa_Status.FIFOError                   // No FIFO error
	        THEN
	            REGION 3.5 – Message preparation

	                // Message composing according to the structure: STX,message body,ETX
	                #ss_MessageP1 := CONCAT(IN1 := #cc_STX,
	                                        IN2 := #cs_Length,
	                                        IN3 := #cs_MessageType,
	                                        IN4 := #ss_LLCSystemID,
	                                        IN5 := "DB_GIN".GIN[#ii_Gin].FedEx.ADCSystemID,
	                                        IN6 := "DB_GIN".GIN[#ii_Gin].FedEx.ImageID,
	                                        IN7 := #ss_PackageID,
	                                        IN8 := "DB_GIN".GIN[#ii_Gin].FedEx.HLCPackageID,
	                                        IN9 := "DB_GIN".GIN[#ii_Gin].FedEx.DIMSystemID,
	                                        IN10 := "DB_GIN".GIN[#ii_Gin].FedEx.DIMStatus,
	                                        IN11 := "DB_GIN".GIN[#ii_Gin].FedEx.PackageDimLength,
	                                        IN12 := "DB_GIN".GIN[#ii_Gin].FedEx.PackageDimWidth,
	                                        IN13 := "DB_GIN".GIN[#ii_Gin].FedEx.PackageDimHeight,
	                                        IN14 := #ss_Gap,
	                                        IN15 := "DB_GIN".GIN[#ii_Gin].FedEx.DIMUOM,
	                                        IN16 := "DB_GIN".GIN[#ii_Gin].FedEx.DimLFTstatusCode,
	                                        IN17 := "DB_GIN".GIN[#ii_Gin].FedEx.AlibiDims,
	                                        IN18 := "DB_GIN".GIN[#ii_Gin].FedEx.SCLSystemID,
	                                        IN19 := "DB_GIN".GIN[#ii_Gin].FedEx.SCLStatus,
	                                        IN20 := "DB_GIN".GIN[#ii_Gin].FedEx.SCLWT,
	                                        IN21 := "DB_GIN".GIN[#ii_Gin].FedEx.SCLWTUOM,
	                                        IN22 := "DB_GIN".GIN[#ii_Gin].FedEx.SCLLFTStatusCode,
	                                        IN23 := "DB_GIN".GIN[#ii_Gin].FedEx.AlibiWeight,
	                                        IN24 := "DB_GIN".GIN[#ii_Gin].FedEx.CellNumber,
	                                        IN25 := "DB_GIN".GIN[#ii_Gin].FedEx.CellsOccupied,
	                                        IN26 := "DB_Time".Timestamp,
	                                        IN27 := #iUDT_Facility.TimeZoneDesignator);

	                #ss_MessageP2 := CONCAT(IN1 := "DB_GIN".GIN[#ii_Gin].FedEx.PackageDataTruncated,
	                                        IN2 := "DB_GIN".GIN[#ii_Gin].FedEx.TotalBarcodeDataLength,
	                                        IN3 := "DB_GIN".GIN[#ii_Gin].FedEx.Barcode1Identification,
	                                        IN4 := "DB_GIN".GIN[#ii_Gin].FedEx.Barcode1status,
	                                        IN5 := "DB_GIN".GIN[#ii_Gin].FedEx.Barcode1datalength,
	                                        IN6 := "DB_GIN".GIN[#ii_Gin].FedEx.Barcode1data,
	                                        IN7 := "DB_GIN".GIN[#ii_Gin].FedEx.Barcode2Identification,
	                                        IN8 := "DB_GIN".GIN[#ii_Gin].FedEx.Barcode2status,
	                                        IN9 := "DB_GIN".GIN[#ii_Gin].FedEx.Barcode2datalength,
	                                        IN10 := "DB_GIN".GIN[#ii_Gin].FedEx.Barcode2data,
	                                        IN11 := "DB_GIN".GIN[#ii_Gin].FedEx.Barcode3Identification,
	                                        IN12 := "DB_GIN".GIN[#ii_Gin].FedEx.Barcode3status,
	                                        IN13 := "DB_GIN".GIN[#ii_Gin].FedEx.Barcode3datalength,
	                                        IN14 := "DB_GIN".GIN[#ii_Gin].FedEx.Barcode3data,
	                                        IN15 := #cc_ETX);

	            END_REGION

	            REGION 3.6 – Maximum number of the message characters

	                #si_MaxMsgLen := "FC_GetNrOfArrayEl"(iv_Array := #sUDT_MessageArray.Character);

	            END_REGION

	            REGION 3.7 – Length of the complete message

	                #si_MsgLen := LEN(#ss_MessageP1) + LEN(#ss_MessageP2);

	                // Message length validation
	                #sa_Status.InvalidMessageLength := #si_MsgLen - 2 <> STRING_TO_INT(#cs_Length);

	            END_REGION

	            REGION 3.8 –  Message array size validation

	                #sa_Status.InvalidMsgArraySize := #si_MsgLen > #si_MaxMsgLen;

	            END_REGION

	            REGION 3.9 –  Message character string conversion to a message array of characters

	                IF (NOT #sa_Status.InvalidMsgArraySize)     // Message character array size is valid
	                THEN

	                    Strg_TO_Chars(Strg := #ss_MessageP1,
	                                  pChars := 0,
	                                  Cnt => #sui_ArrayOffset,
	                                  Chars := #sUDT_MessageArray.Character);

	                    Strg_TO_Chars(Strg := #ss_MessageP2,
	                                  pChars := #sui_ArrayOffset,
	                                  Cnt => #sui_MsgArrayElNr,
	                                  Chars := #sUDT_MessageArray.Character);

	                END_IF;

	            END_REGION

	            REGION 3.10 – Clearing remaining characters in the message character array

	                IF (NOT #sa_Status.InvalidMsgArraySize)     // Message character array size is valid
	                THEN

	                    // Filling up not used message character array elements with '$00' (ASCII - 16#00)
	                    FILL_BLK(IN := #cc_NULL,                                                                             // Fill not used message char array elements with '$00'
	                             COUNT := UINT_TO_ULINT(INT_TO_UINT(#si_MaxMsgLen) - #sui_MsgArrayElNr - #sui_ArrayOffset),
	                             OUT => #sUDT_MessageArray.Character[#sui_MsgArrayElNr + #sui_ArrayOffset]);

	                END_IF;

	            END_REGION

	            REGION 3.11 – Message write into a FIFO register

	                IF NOT #sa_Status.InvalidMsgArraySize           // Message character array size is valid
	                    AND NOT #sa_Status.InvalidMessageLength     // Message length is valid
	                THEN

	                    // Mode 'W' - Write FIFO record
	                    "FC_Fifo"(ic_Mode := 'W',
	                              qUDT_Status => #sa_Status.FIFOStatus,
	                              qx_Error => #sa_Status.FIFOError,
	                              qx_Warning => #sa_Status.FIFOWarning,
	                              iqv_Data := #sUDT_MessageArray,

	                              iqUDT_FifoHeader := #iqUDT_FifoHeader,
	                              iqv_DataBuffer := #iqa_FifoData);

	                ELSE
	                    // Increase counter messages not sent because of wrong message length
	                    #sa_Statistics.NotSentWrongMsgLen += 1;

	                END_IF;

	            END_REGION
	            #si_OldGin := #ii_Gin;


	        END_IF;

	        // In case of FIFO full, the FIFO full error bit and FIFO collective error bit are set
	    ELSE
	        #sa_Status.FIFOError := TRUE;
	        #sa_Status.FIFOStatus.FifoFull := TRUE;

	    END_IF;

	END_REGION

	REGION 4 - Writing outputs

	    #sx_Error := #sa_Status.InvalidMessageLength        // Invalid message length
	    OR #sa_Status.InvalidGIN                            // Invalid GIN
	    OR #sa_Status.InvalidMsgArraySize                   // Invalid message array size
	    OR #sa_Status.FIFOError;                            // FIFO error

	END_REGION

	REGION 5 Unexpected DL Request

	    IF #iqx_UnexpectedDLReq THEN
	        REGION 5.1 – FIFO header status update

	            // Mode 'S' - FIFO register status update
	            "FC_Fifo"(ic_Mode := 'S',
	                      qUDT_Status => #sa_Status.FIFOStatus,
	                      qx_Error => #sa_Status.FIFOError,
	                      qx_Warning => #sa_Status.FIFOWarning,
	                      iqv_Data := #sUDT_MessageArray,
	                      iqUDT_FifoHeader := #iqUDT_FifoHeader,
	                      iqv_DataBuffer := #iqa_FifoData);
	        END_REGION

	        REGION 5.2 – Message preparation
	            IF NOT #iqUDT_FifoHeader.Status.Full                       // FIFO isn't full
	            THEN

	                REGION Sequential  ID
	                    // ss_SequencialID character string clearing
	                    #ss_SequencialID := '';
	                    // ss_SequencialID integer input conversion to a character string
	                    VAL_STRG(IN := "DB_ExternalGIN".UnexpectedSI.FedEx.CustomerID,
	                             SIZE := 0,
	                             PREC := 0,
	                             FORMAT := 0,
	                             P := 1,
	                             OUT => #ss_SequencialID);
	                    // Length of the ss_SequencialID character string
	                    #si_StringLen := LEN(#ss_SequencialID);

	                    // ss_SequencialID character string leading zeros addition
	                    IF (#si_StringLen < 6)
	                    THEN
	                        FOR #si_LenFillLoop := 1 TO 6 - #si_StringLen DO
	                            #ss_SequencialID := CONCAT(IN1 := '0',
	                                                       IN2 := #ss_SequencialID);
	                        END_FOR;
	                    END_IF;
	                END_REGION

	                REGION LLC System ID
	                    // Build LLC Syatem ID
	                    #ss_LLCSystemID := CONCAT(IN1 := #is_DEPCOD,
	                                              IN2 := #is_LOConEquipment,
	                                              IN3 := #is_TYPofEquipment,
	                                              IN4 := #is_NumberOfTheEquipment);

	                END_REGION

	                REGION Package ID
	                    // Build Package ID
	                    #ss_PackageID := CONCAT(IN1 := #is_TrayCellNumber,
	                                            IN2 := #is_SorterNumber,
	                                            IN3 := #is_InductionNumber,
	                                            IN4 := #is_AreaNumber,
	                                            IN5 := #ss_SequencialID);
	                END_REGION

	                REGION Gap

	                    #ss_Gap := '000';

	                END_REGION

	                IF NOT #sa_Status.FIFOError                   // No FIFO error
	                THEN
	                    REGION Message preparation

	                        #ss_MessageP1 := CONCAT(IN1 := #cc_STX,
	                                                IN2 := #cs_Length,
	                                                IN3 := #cs_MessageType,
	                                                IN4 := #ss_LLCSystemID,
	                                                IN5 := "DB_ExternalGIN".UnexpectedSI.FedEx.ADCSystemID,
	                                                IN6 := "DB_ExternalGIN".UnexpectedSI.FedEx.ImageID,
	                                                IN7 := "DB_ExternalGIN".UnexpectedSI.FedEx.PackageID,
	                                                IN8 := "DB_ExternalGIN".UnexpectedSI.FedEx.HLCPackageID,
	                                                IN9 := "DB_ExternalGIN".UnexpectedSI.FedEx.DIMSystemID,
	                                                IN10 := "DB_ExternalGIN".UnexpectedSI.FedEx.DIMStatus,
	                                                IN11 := "DB_ExternalGIN".UnexpectedSI.FedEx.PackageDimLength,
	                                                IN12 := "DB_ExternalGIN".UnexpectedSI.FedEx.PackageDimWidth,
	                                                IN13 := "DB_ExternalGIN".UnexpectedSI.FedEx.PackageDimHeight,
	                                                IN14 := #ss_Gap,
	                                                IN15 := "DB_ExternalGIN".UnexpectedSI.FedEx.DIMUOM,
	                                                IN16 := "DB_ExternalGIN".UnexpectedSI.FedEx.DimLFTstatusCode,
	                                                IN17 := "DB_ExternalGIN".UnexpectedSI.FedEx.AlibiDims,
	                                                IN18 := "DB_ExternalGIN".UnexpectedSI.FedEx.SCLSystemID,
	                                                IN19 := "DB_ExternalGIN".UnexpectedSI.FedEx.SCLStatus,
	                                                IN20 := "DB_ExternalGIN".UnexpectedSI.FedEx.SCLWT,
	                                                IN21 := "DB_ExternalGIN".UnexpectedSI.FedEx.SCLWTUOM,
	                                                IN22 := "DB_ExternalGIN".UnexpectedSI.FedEx.SCLLFTStatusCode,
	                                                IN23 := "DB_ExternalGIN".UnexpectedSI.FedEx.AlibiWeight,
	                                                IN24 := "DB_ExternalGIN".UnexpectedSI.FedEx.CellNumber,
	                                                IN25 := "DB_ExternalGIN".UnexpectedSI.FedEx.CellsOccupied,
	                                                IN26 := "DB_Time".Timestamp,
	                                                IN27 := #iUDT_Facility.TimeZoneDesignator);

	                        #ss_MessageP2 := CONCAT(IN1 := "DB_ExternalGIN".UnexpectedSI.FedEx.PackageDataTruncated,
	                                                IN2 := "DB_ExternalGIN".UnexpectedSI.FedEx.TotalBarcodeDataLength,
	                                                IN3 := "DB_ExternalGIN".UnexpectedSI.FedEx.Barcode1Identification,
	                                                IN4 := "DB_ExternalGIN".UnexpectedSI.FedEx.Barcode1status,
	                                                IN5 := "DB_ExternalGIN".UnexpectedSI.FedEx.Barcode1datalength,
	                                                IN6 := "DB_ExternalGIN".UnexpectedSI.FedEx.Barcode1data,
	                                                IN7 := "DB_ExternalGIN".UnexpectedSI.FedEx.Barcode2Identification,
	                                                IN8 := "DB_ExternalGIN".UnexpectedSI.FedEx.Barcode2status,
	                                                IN9 := "DB_ExternalGIN".UnexpectedSI.FedEx.Barcode2datalength,
	                                                IN10 := "DB_ExternalGIN".UnexpectedSI.FedEx.Barcode2data,
	                                                IN11 := "DB_ExternalGIN".UnexpectedSI.FedEx.Barcode3Identification,
	                                                IN12 := "DB_ExternalGIN".UnexpectedSI.FedEx.Barcode3status,
	                                                IN13 := "DB_ExternalGIN".UnexpectedSI.FedEx.Barcode3datalength,
	                                                IN14 := "DB_ExternalGIN".UnexpectedSI.FedEx.Barcode3data,
	                                                IN15 := #cc_ETX);

	                    END_REGION

	                    REGION Maximum number of the message characters

	                        #si_MaxMsgLen := "FC_GetNrOfArrayEl"(iv_Array := #sUDT_MessageArray.Character);

	                    END_REGION

	                    REGION Length of the complete message

	                        #si_MsgLen := LEN(#ss_MessageP1) + LEN(#ss_MessageP2);

	                        // Message length validation
	                        #sa_Status.InvalidMessageLength := #si_MsgLen - 2 <> STRING_TO_INT(#cs_Length);

	                    END_REGION

	                    REGION Message array size validation

	                        #sa_Status.InvalidMsgArraySize := #si_MsgLen > #si_MaxMsgLen;

	                    END_REGION

	                    REGION Message character string conversion to a message array of characters

	                        IF (NOT #sa_Status.InvalidMsgArraySize)     // Message character array size is valid
	                        THEN

	                            Strg_TO_Chars(Strg := #ss_MessageP1,
	                                          pChars := 0,
	                                          Cnt => #sui_ArrayOffset,
	                                          Chars := #sUDT_MessageArray.Character);

	                            Strg_TO_Chars(Strg := #ss_MessageP2,
	                                          pChars := #sui_ArrayOffset,
	                                          Cnt => #sui_MsgArrayElNr,
	                                          Chars := #sUDT_MessageArray.Character);

	                        END_IF;

	                    END_REGION

	                    REGION Clearing remaining characters in the message character array

	                        IF (NOT #sa_Status.InvalidMsgArraySize)     // Message character array size is valid
	                        THEN

	                            // Filling up not used message character array elements with '$00' (ASCII - 16#00)
	                            FILL_BLK(IN := #cc_NULL,                                                                             // Fill not used message char array elements with '$00'
	                                     COUNT := UINT_TO_ULINT(INT_TO_UINT(#si_MaxMsgLen) - #sui_MsgArrayElNr - #sui_ArrayOffset),
	                                     OUT => #sUDT_MessageArray.Character[#sui_MsgArrayElNr + #sui_ArrayOffset]);

	                        END_IF;

	                    END_REGION

	                    REGION Message write into a FIFO register

	                        IF NOT #sa_Status.InvalidMsgArraySize           // Message character array size is valid
	                            AND NOT #sa_Status.InvalidMessageLength     // Message length is valid
	                        THEN

	                            // Mode 'W' - Write FIFO record
	                            "FC_Fifo"(ic_Mode := 'W',
	                                      qUDT_Status => #sa_Status.FIFOStatus,
	                                      qx_Error => #sa_Status.FIFOError,
	                                      qx_Warning => #sa_Status.FIFOWarning,
	                                      iqv_Data := #sUDT_MessageArray,
	                                      iqUDT_FifoHeader := #iqUDT_FifoHeader,
	                                      iqv_DataBuffer := #iqa_FifoData);

	                        ELSE
	                            // Increase counter messages not sent because of wrong message length
	                            #sa_Statistics.NotSentWrongMsgLen += 1;

	                        END_IF;

	                    END_REGION
	                    #iqx_UnexpectedDLReq := FALSE;

	                END_IF;

	                // In case of FIFO full, the FIFO full error bit and FIFO collective error bit are set
	            ELSE
	                #sa_Status.FIFOError := TRUE;
	                #sa_Status.FIFOStatus.FifoFull := TRUE;

	            END_IF;

	        END_REGION
	    END_IF;

	END_REGION

	REGION 6 - Writing outputs

	    #qx_Error := #sa_Status.InvalidMessageLength        // Invalid message length
	    OR #sa_Status.InvalidGIN                            // Invalid GIN
	    OR #sa_Status.InvalidMsgArraySize                   // Invalid message array size
	    OR #sa_Status.FIFOError                             // FIFO error
	    OR #sx_Error;

	END_REGION

END_FUNCTION_BLOCK

FUNCTION_BLOCK "FB_FedExDivertVerificationMessage"
TITLE = FB_Heartbeat
{ S7_Optimized_Access := 'TRUE' }
AUTHOR : MHSE
FAMILY : UPS_SpecificCommunication
VERSION : 3.0
// ATTRIBUTES
// AUTO_NUMBER = True
// BLOCK_NUMBER = 68
// END_ATTRIBUTES
//Function block to send and monitor the UPS heartbeat message.
   VAR_INPUT
      iUDT_Facility { ExternalAccessible := 'False'; ExternalVisible := 'False'; ExternalWritable := 'False'} : "UDT_FedExFacility";   // System configuration
      is_LOConEquipment { ExternalAccessible := 'False'; ExternalVisible := 'False'; ExternalWritable := 'False'} : String[3];   // Location of the equipment
      is_DEPCOD { ExternalAccessible := 'False'; ExternalVisible := 'False'; ExternalWritable := 'False'} : String[6];   // Depot Code
      is_TYPofEquipment { ExternalAccessible := 'False'; ExternalVisible := 'False'; ExternalWritable := 'False'} : String[3];   // Type of equipment
      is_NumberOfTheEquipment { ExternalAccessible := 'False'; ExternalVisible := 'False'; ExternalWritable := 'False'} : String[3];   // Number of the equipment 001-999
      is_TrayCellNumber { ExternalAccessible := 'False'; ExternalVisible := 'False'; ExternalWritable := 'False'} : String[3];   // Tray/Cell number (for loop sorters) or generated by LLC (on line sorters).
      is_SorterNumber { ExternalAccessible := 'False'; ExternalVisible := 'False'; ExternalWritable := 'False'} : String[2];   // Sorter number
      is_InductionNumber { ExternalAccessible := 'False'; ExternalVisible := 'False'; ExternalWritable := 'False'} : String[2];   // Induction number
      is_AreaNumber { ExternalAccessible := 'False'; ExternalVisible := 'False'; ExternalWritable := 'False'} : String[2];   // Area number
      ii_Gin { ExternalAccessible := 'False'; ExternalVisible := 'False'; ExternalWritable := 'False'} : Int;   // GIN number
   END_VAR

   VAR_OUTPUT
      qx_Error { ExternalAccessible := 'False'; ExternalVisible := 'False'; ExternalWritable := 'False'} : Bool;   // Error
   END_VAR

   VAR_IN_OUT
      iqUDT_FifoHeader : "UDT_FifoHeader";   // FIFO header
      iqa_FifoData : Array[*] of "UDT_Message";   // FIFO data
   END_VAR

   VAR
      sUDT_MessageArray { ExternalAccessible := 'False'; ExternalVisible := 'False'; ExternalWritable := 'False'; S7_SetPoint := 'False'} : "UDT_Message";   // Message character array
      ss_Status { ExternalAccessible := 'False'; ExternalVisible := 'False'; ExternalWritable := 'False'} : Struct   // Status structure
         FIFOStatus { ExternalAccessible := 'False'; ExternalVisible := 'False'; ExternalWritable := 'False'} : "UDT_FifoStatus";   // FIFO status structure
         FIFOError { ExternalAccessible := 'False'; ExternalVisible := 'False'; ExternalWritable := 'False'; S7_SetPoint := 'True'} : Bool;   // FIFO data buffer full
         FIFOWarning { ExternalAccessible := 'False'; ExternalVisible := 'False'; ExternalWritable := 'False'; S7_SetPoint := 'True'} : Bool;   // FIFO error
         InvalidGIN { ExternalAccessible := 'False'; ExternalVisible := 'False'; ExternalWritable := 'False'} : Bool;   //  Invalid GIN
         InvalidMessageLength { ExternalAccessible := 'False'; ExternalVisible := 'False'; ExternalWritable := 'False'} : Bool;   // Calculated message length is different than required
         InvalidMsgArraySize { ExternalAccessible := 'False'; ExternalVisible := 'False'; ExternalWritable := 'False'} : Bool;   // Length of the message is bigger than length of message array
      END_STRUCT;
      ss_Statistics { ExternalAccessible := 'False'; ExternalVisible := 'False'; ExternalWritable := 'False'} : Struct   // Statistics structure
         NotSentWrongMsgLen { ExternalAccessible := 'False'; ExternalVisible := 'False'; ExternalWritable := 'False'} : DInt;   // COMISSIONING PURPOSE Messages not sent because built message length does not match with required message length
      END_STRUCT;
      ss_LLCSystemID { ExternalAccessible := 'False'; ExternalVisible := 'False'; ExternalWritable := 'False'} : String[15];   // Identifier of Low-Level controls
      ss_SequencialID { ExternalAccessible := 'False'; ExternalVisible := 'False'; ExternalWritable := 'False'} : String[6];   // Identifier of Low-Level controls
      ss_Message { ExternalAccessible := 'False'; ExternalVisible := 'False'; ExternalWritable := 'False'} : String;   // Message character string
      ss_PackageID { ExternalAccessible := 'False'; ExternalVisible := 'False'; ExternalWritable := 'False'} : String[15];   // Identifier of Low-Level controls
      ss_Recirculation { ExternalAccessible := 'False'; ExternalVisible := 'False'; ExternalWritable := 'False'} : String[2];   // Converted to string
      sui_MsgArrayElNr { ExternalAccessible := 'False'; ExternalVisible := 'False'; ExternalWritable := 'False'} : UInt;   // Invalid message array size
      sui_ArrayOffset { ExternalAccessible := 'False'; ExternalVisible := 'False'; ExternalWritable := 'False'} : UInt;   // Offset for writing in the array
      si_OldGin { ExternalAccessible := 'False'; ExternalVisible := 'False'; ExternalWritable := 'False'} : Int;   // Previous Gin
      si_StringLen { ExternalAccessible := 'False'; ExternalVisible := 'False'; ExternalWritable := 'False'} : Int;   // Length of string used in loops to pad string with spaces or 0
      si_LenFillLoop { ExternalAccessible := 'False'; ExternalVisible := 'False'; ExternalWritable := 'False'} : Int;   // Loop couter
      si_MaxMsgLen { ExternalAccessible := 'False'; ExternalVisible := 'False'; ExternalWritable := 'False'} : Int;   // Maximum message length
      si_MsgLen { ExternalAccessible := 'False'; ExternalVisible := 'False'; ExternalWritable := 'False'} : Int;   // String character message length
   END_VAR

   VAR_TEMP
      tw_HTA_RET_VAL : Word;
   END_VAR

   VAR CONSTANT
      cc_NULL : Char := '$00';   // NULL sign
      cc_STX : Char := '$02';   // Start of the text
      cc_ETX : String := '$03';   // End of the text
      cs_Length : String := '0180';   // Legth of the message
      cs_MessageType : String := 'DV';   // Message type
   END_VAR


BEGIN
	(*
	----------------------------------------------------------------------------------------

	Version history:
	Date        | Version   | Author        | Remark
	----------------------------------------------------------------------------------------
	29/06/2021  | 1.0       | F.Baten       | first release MHS TIA 16.0
	10/11/2021  | 1.2       | M.Piela       | Updating regions numbering
	05/04/2022  | 1.3       | K.Pokorski    | Review
	21/02/2023  | 4.0       | F.Baten       | 4.0 Release TIA 17.5
	*)

	REGION 1 – FIFO header status update

	    // Mode 'S' - FIFO register status update
	    "FC_Fifo"(ic_Mode := 'S',
	              qUDT_Status => #ss_Status.FIFOStatus,
	              qx_Error => #ss_Status.FIFOError,
	              qx_Warning => #ss_Status.FIFOWarning,
	              iqv_Data := #sUDT_MessageArray,
	              iqUDT_FifoHeader := #iqUDT_FifoHeader,
	              iqv_DataBuffer := #iqa_FifoData);
	END_REGION

	REGION 2 - GIN validation

	    // GIN validation
	    #ss_Status.InvalidGIN :=
	    #ii_Gin < 1
	    OR #ii_Gin > 9999;

	END_REGION

	REGION 3 – Message preparation

	    IF NOT #iqUDT_FifoHeader.Status.Full               // FIFO isn't full
	    THEN
	        IF #ii_Gin <> #si_OldGin                            // New gin is different than old
	            AND NOT #ss_Status.InvalidGIN                   // Gin is valid
	        THEN
	            REGION 3.1 - Sequencial ID
	                // ss_SequencialID character string clearing
	                #ss_SequencialID := '';
	                // ss_SequencialID integer input conversion to a character string
	                VAL_STRG(IN := "DB_GIN".GIN[#ii_Gin].FedEx.CustomerID,
	                         SIZE := 0,
	                         PREC := 0,
	                         FORMAT := 0,
	                         P := 1,
	                         OUT => #ss_SequencialID);
	                // Length of the ss_SequencialID character string
	                #si_StringLen := LEN(#ss_SequencialID);

	                // ss_SequencialID character string leading zeros addition
	                IF (#si_StringLen < 6)
	                THEN
	                    FOR #si_LenFillLoop := 1 TO 6 - #si_StringLen DO
	                        #ss_SequencialID := CONCAT(IN1 := '0',
	                                                   IN2 := #ss_SequencialID);
	                    END_FOR;
	                END_IF;
	            END_REGION

	            REGION 3.2 LLC Syatem ID
	                // Build LLC Syatem ID
	                #ss_LLCSystemID := CONCAT(IN1 := #is_DEPCOD,
	                                          IN2 := #is_LOConEquipment,
	                                          IN3 := #is_TYPofEquipment,
	                                          IN4 := #is_NumberOfTheEquipment);

	            END_REGION

	            REGION 3.3 - Package ID
	                // Build Package ID
	                #ss_PackageID := CONCAT(IN1 := #is_TrayCellNumber,
	                                        IN2 := #is_SorterNumber,
	                                        IN3 := #is_InductionNumber,
	                                        IN4 := #is_AreaNumber,
	                                        IN5 := #ss_SequencialID);
	            END_REGION

	            REGION 3.4 - Number of recirculation
	                // Character string clearing
	                #ss_Recirculation := '';
	                // integer input conversion to a character string
	                VAL_STRG(IN := "DB_GIN".GIN[#ii_Gin].General.NrOfRecirculations,
	                         SIZE := 0,
	                         PREC := 0,
	                         FORMAT := 0,
	                         P := 1,
	                         OUT => #ss_Recirculation);
	                // Length of the gap character string
	                #si_StringLen := LEN(#ss_Recirculation);
	                // Gap character string leading zeros addition
	                IF (#si_StringLen < 2)
	                THEN
	                    #ss_Recirculation := CONCAT(IN1 := '0',
	                                                IN2 := #ss_Recirculation);
	                END_IF;

	            END_REGION

	            REGION 3.5 – Message preparation
	                // Message composing according to the structure: STX,message body,ETX
	                #ss_Message := CONCAT(IN1 := #cc_STX,
	                                      IN2 := #cs_Length,
	                                      IN3 := #cs_MessageType,
	                                      IN4 := #ss_LLCSystemID,
	                                      IN5 := #ss_PackageID,
	                                      IN6 := "DB_GIN".GIN[#ii_Gin].FedEx.HLCPackageID,
	                                      IN7 := "DB_GIN".GIN[#ii_Gin].FedEx.CellNumber,
	                                      IN8 := "DB_GIN".GIN[#ii_Gin].FedEx.ActualDestination,
	                                      IN9 := "DB_GIN".GIN[#ii_Gin].FedEx.PackageEntrancePoint,
	                                      IN10 := "DB_GIN".GIN[#ii_Gin].FedEx.PackageEntranceState,
	                                      IN11 := "DB_GIN".GIN[#ii_Gin].FedEx.PackageExitPoint,
	                                      IN12 := "DB_GIN".GIN[#ii_Gin].FedEx.PackageExitState,
	                                      IN13 := "DB_GIN".GIN[#ii_Gin].FedEx.Destination1,
	                                      IN14 := "DB_GIN".GIN[#ii_Gin].FedEx.ReasonCode1,
	                                      IN15 := "DB_GIN".GIN[#ii_Gin].FedEx.Destination2,
	                                      IN16 := "DB_GIN".GIN[#ii_Gin].FedEx.ReasonCode2,
	                                      IN17 := "DB_GIN".GIN[#ii_Gin].FedEx.Destination3,
	                                      IN18 := "DB_GIN".GIN[#ii_Gin].FedEx.ReasonCode3,
	                                      IN19 := "DB_GIN".GIN[#ii_Gin].FedEx.Destination4,
	                                      IN20 := "DB_GIN".GIN[#ii_Gin].FedEx.ReasonCode4,
	                                      IN21 := "DB_GIN".GIN[#ii_Gin].FedEx.Destination5,
	                                      IN22 := "DB_GIN".GIN[#ii_Gin].FedEx.ReasonCode5,
	                                      IN23 := #ss_Recirculation,
	                                      IN24 := "DB_Time".Timestamp,
	                                      IN25 := #iUDT_Facility.TimeZoneDesignator,
	                                      IN26 := #cc_ETX);
	            END_REGION

	            REGION 3.6 – Maximum number of the message characters

	                #si_MaxMsgLen := "FC_GetNrOfArrayEl"(iv_Array := #sUDT_MessageArray.Character);

	            END_REGION

	            REGION 3.7 – Length of the complete message

	                #si_MsgLen := LEN(#ss_Message);

	                // Message length validation
	                #ss_Status.InvalidMessageLength := #si_MsgLen - 2 <> STRING_TO_INT(#cs_Length);

	            END_REGION

	            REGION 3.8 –  Message array size validation

	                #ss_Status.InvalidMsgArraySize := #si_MsgLen > #si_MaxMsgLen;

	            END_REGION

	            REGION 3.9 –  Message character string conversion to a message array of characters

	                IF (NOT #ss_Status.InvalidMsgArraySize)     // Message character array size is valid
	                THEN

	                    Strg_TO_Chars(Strg := #ss_Message,
	                                  pChars := 0,
	                                  Cnt => #sui_MsgArrayElNr,
	                                  Chars := #sUDT_MessageArray.Character);
	                END_IF;

	            END_REGION

	            REGION 3.10 – Clearing remaining characters in the message character array

	                IF (NOT #ss_Status.InvalidMsgArraySize)     // Message character array size is valid
	                THEN

	                    // Filling up not used message character array elements with '$00' (ASCII - 16#00)
	                    FILL_BLK(IN := #cc_NULL,                                                                             // Fill not used message char array elements with '$00'
	                             COUNT := UINT_TO_ULINT(INT_TO_UINT(#si_MaxMsgLen) - #sui_MsgArrayElNr - #sui_ArrayOffset),
	                             OUT => #sUDT_MessageArray.Character[#sui_MsgArrayElNr + #sui_ArrayOffset]);

	                END_IF;

	            END_REGION

	            REGION 3.11 – Message write into a FIFO register

	                IF NOT #ss_Status.InvalidMsgArraySize               // Message character array size is valid
	                    AND NOT #ss_Status.InvalidMessageLength         //Message length is valid
	                THEN

	                    // Mode 'W' - Write FIFO record
	                    "FC_Fifo"(ic_Mode := 'W',
	                              qUDT_Status => #ss_Status.FIFOStatus,
	                              qx_Error => #ss_Status.FIFOError,
	                              qx_Warning => #ss_Status.FIFOWarning,
	                              iqv_Data := #sUDT_MessageArray,
	                              iqUDT_FifoHeader := #iqUDT_FifoHeader,
	                              iqv_DataBuffer := #iqa_FifoData);
	                ELSE
	                    // Increase counter messages not sent because of wrong message length
	                    #ss_Statistics.NotSentWrongMsgLen += 1;

	                END_IF;

	            END_REGION
	            #si_OldGin := #ii_Gin;
	        END_IF;

	        // In case of FIFO full, the FIFO full error bit and FIFO collective error bit are set
	    ELSE
	        #ss_Status.FIFOError := TRUE;
	        #ss_Status.FIFOStatus.FifoFull := TRUE;

	    END_IF;

	END_REGION

	REGION 4 - Writing outputs

	    #qx_Error := #ss_Status.InvalidMessageLength        // Invalid message length
	    OR #ss_Status.InvalidGIN                            // Invalid GIN
	    OR #ss_Status.InvalidMsgArraySize                   // Invalid message array size
	    OR #ss_Status.FIFOError;                            // FIFO error

	END_REGION
END_FUNCTION_BLOCK

FUNCTION_BLOCK "FB_FedExDVLost"
{ S7_Optimized_Access := 'TRUE' }
VERSION : 0.1
// ATTRIBUTES
// AUTO_NUMBER = True
// BLOCK_NUMBER = 69
// END_ATTRIBUTES
   VAR_INPUT
      is_PackageExitPoint { ExternalAccessible := 'False'; ExternalVisible := 'False'; ExternalWritable := 'False'} : String[14];
      is_RejectChute { ExternalAccessible := 'False'; ExternalVisible := 'False'; ExternalWritable := 'False'} : String[6];
   END_VAR

   VAR_IN_OUT
      iqa_FifoLostGinData : Array[*] of Int;   // Fifo data
      iqUDT_FifoLostGinHeader : "UDT_FifoHeader";   // Fifo header
      iqi_GINDVMessageLost { ExternalAccessible := 'False'; ExternalVisible := 'False'; ExternalWritable := 'False'} : Int;   // GIN number
   END_VAR

   VAR
      ss_Status { ExternalAccessible := 'False'; ExternalVisible := 'False'; ExternalWritable := 'False'} : Struct   // Fifo status
         FIFOStatus { ExternalAccessible := 'False'; ExternalVisible := 'False'; ExternalWritable := 'False'; S7_SetPoint := 'False'} : "UDT_FifoStatus";
         FIFOError { ExternalAccessible := 'False'; ExternalVisible := 'False'; ExternalWritable := 'False'; S7_SetPoint := 'True'} : Bool;
         FIFOWarning { ExternalAccessible := 'False'; ExternalVisible := 'False'; ExternalWritable := 'False'} : Bool;
         InvalidGIN { ExternalAccessible := 'False'; ExternalVisible := 'False'; ExternalWritable := 'False'} : Bool;
         InvalidMessageLength { ExternalAccessible := 'False'; ExternalVisible := 'False'; ExternalWritable := 'False'} : Bool;
         InvalidMsgArraySize { ExternalAccessible := 'False'; ExternalVisible := 'False'; ExternalWritable := 'False'} : Bool;
      END_STRUCT;
   END_VAR

   VAR_TEMP
      ti_GIN : Int;
   END_VAR


BEGIN
	(*
	----------------------------------------------------------------------------------------

	Version history:
	Date        | Version   | Author        | Remark
	----------------------------------------------------------------------------------------
	26/04/2022  | 1.0       | K. Pokorski   | first release MHS TIA 16.0
	21/02/2023  | 4.0       | F.Baten       | 4.0 Release TIA 17.5
	13/03/2024  | 4.1       | S. Nieświec   | 4.1 Release TIA 18
	*)
	REGION 1 - Read fifo status

	    "FC_Fifo"(ic_Mode := 'S',
	              qUDT_Status => #ss_Status.FIFOStatus,
	              qx_Error => #ss_Status.FIFOError,
	              qx_Warning => #ss_Status.FIFOWarning,
	              iqv_Data := #ti_GIN,
	              iqUDT_FifoHeader := #iqUDT_FifoLostGinHeader,
	              iqv_DataBuffer := #iqa_FifoLostGinData);
	END_REGION

	REGION 2 - Read first lost GIN

	    IF (NOT #iqUDT_FifoLostGinHeader.Status.Empty                             // FIFO not empty
	        AND NOT #ss_Status.FIFOError)                                      // No FIFO error
	    THEN

	        // Mode 'R' - Read FIFO record
	        "FC_Fifo"(ic_Mode := 'R',
	                  qUDT_Status => #ss_Status.FIFOStatus,
	                  qx_Error => #ss_Status.FIFOError,
	                  qx_Warning => #ss_Status.FIFOWarning,
	                  iqv_Data := #ti_GIN,
	                  iqUDT_FifoHeader := #iqUDT_FifoLostGinHeader,
	                  iqv_DataBuffer := #iqa_FifoLostGinData);

	        "DB_GIN".GIN[#ti_GIN].General.Lost := TRUE;
	        "DB_GIN".GIN[#ti_GIN].FedEx.ReasonCode1 := '00000800';
	        "DB_GIN".GIN[#ti_GIN].FedEx.PackageExitPoint := #is_PackageExitPoint;
	        "DB_GIN".GIN[#ti_GIN].FedEx.PackageExitState := '2';
	        "DB_GIN".GIN[#ti_GIN].FedEx.ActualDestination := #is_RejectChute;
	        #iqi_GINDVMessageLost := #ti_GIN;

	    END_IF;
	END_REGION


END_FUNCTION_BLOCK

FUNCTION_BLOCK "FB_FedExDXMessage"
TITLE = FB_Heartbeat
{ S7_Optimized_Access := 'TRUE' }
AUTHOR : MHSE
FAMILY : UPS_SpecificCommunication
VERSION : 3.0
// ATTRIBUTES
// AUTO_NUMBER = True
// BLOCK_NUMBER = 70
// END_ATTRIBUTES
//Function block to send and monitor the UPS heartbeat message.
   VAR_INPUT
      iUDT_Facility { ExternalAccessible := 'False'; ExternalVisible := 'False'; ExternalWritable := 'False'} : "UDT_FedExFacility";   // System configuration
      is_LOConEquipment { ExternalAccessible := 'False'; ExternalVisible := 'False'; ExternalWritable := 'False'} : String[3];   // Location of the equipment
      is_DEPCOD { ExternalAccessible := 'False'; ExternalVisible := 'False'; ExternalWritable := 'False'} : String[6];   // Depot Code
      is_TYPofEquipment { ExternalAccessible := 'False'; ExternalVisible := 'False'; ExternalWritable := 'False'} : String[3];   // Type of equipment
      is_NumberOfTheEquipment { ExternalAccessible := 'False'; ExternalVisible := 'False'; ExternalWritable := 'False'} : String[3];   // Number of the equipment 001-999
      is_TrayCellNumber { ExternalAccessible := 'False'; ExternalVisible := 'False'; ExternalWritable := 'False'} : String[3];   // Tray/Cell number (for loop sorters) or generated by LLC (on line sorters).
      is_SorterNumber { ExternalAccessible := 'False'; ExternalVisible := 'False'; ExternalWritable := 'False'} : String[2];   // Sorter number
      is_InductionNumber { ExternalAccessible := 'False'; ExternalVisible := 'False'; ExternalWritable := 'False'} : String[2];   // Induction number
      is_AreaNumber { ExternalAccessible := 'False'; ExternalVisible := 'False'; ExternalWritable := 'False'} : String[2];   // Area number
      ii_Gin { ExternalAccessible := 'False'; ExternalVisible := 'False'; ExternalWritable := 'False'} : Int;   // GIN number
   END_VAR

   VAR_OUTPUT
      qx_Error { ExternalAccessible := 'False'; ExternalVisible := 'False'; ExternalWritable := 'False'} : Bool;   // Error
   END_VAR

   VAR_IN_OUT
      iqUDT_FifoHeader : "UDT_FifoHeader";   // FIFO header
      iqa_FifoData : Array[*] of "UDT_Message";   // FIFO data
      iqx_Unexpected_DX_Req { ExternalAccessible := 'False'; ExternalVisible := 'False'; ExternalWritable := 'False'} : Bool;
   END_VAR

   VAR
      sUDT_MessageArray { ExternalAccessible := 'False'; ExternalVisible := 'False'; ExternalWritable := 'False'; S7_SetPoint := 'False'} : "UDT_Message";   // Message character array
      sa_Status { ExternalAccessible := 'False'; ExternalVisible := 'False'; ExternalWritable := 'False'} : Struct   // Status structure
         FIFOStatus { ExternalAccessible := 'False'; ExternalVisible := 'False'; ExternalWritable := 'False'} : "UDT_FifoStatus";   // FIFO status structure
         FIFOError { ExternalAccessible := 'False'; ExternalVisible := 'False'; ExternalWritable := 'False'; S7_SetPoint := 'True'} : Bool;   // FIFO data buffer full
         FIFOWarning { ExternalAccessible := 'False'; ExternalVisible := 'False'; ExternalWritable := 'False'; S7_SetPoint := 'True'} : Bool;   // FIFO error
         InvalidGIN { ExternalAccessible := 'False'; ExternalVisible := 'False'; ExternalWritable := 'False'} : Bool;   //  Invalid GIN
         InvalidMessageLength { ExternalAccessible := 'False'; ExternalVisible := 'False'; ExternalWritable := 'False'} : Bool;   // Calculated message length is different than required
         InvalidMsgArraySize { ExternalAccessible := 'False'; ExternalVisible := 'False'; ExternalWritable := 'False'} : Bool;   // Heartbeat timeout lower than zero or lower than heartbeat time interval
      END_STRUCT;
      sa_Statistics { ExternalAccessible := 'False'; ExternalVisible := 'False'; ExternalWritable := 'False'} : Struct   // Statistics structure
         NotSentWrongMsgLen { ExternalAccessible := 'False'; ExternalVisible := 'False'; ExternalWritable := 'False'} : DInt;   // COMISSIONING PURPOSE Messages not sent because built message length does not match with required message length
      END_STRUCT;
      ss_LLCSystemID { ExternalAccessible := 'False'; ExternalVisible := 'False'; ExternalWritable := 'False'} : String[15];   // Identifier of Low-Level controls
      ss_SequencialID { ExternalAccessible := 'False'; ExternalVisible := 'False'; ExternalWritable := 'False'} : String[6];   // Identifier of Low-Level controls
      ss_MessageP1 { ExternalAccessible := 'False'; ExternalVisible := 'False'; ExternalWritable := 'False'} : String;   // Message character string part 1
      ss_MessageP2 { ExternalAccessible := 'False'; ExternalVisible := 'False'; ExternalWritable := 'False'} : String;   // Message character string part 2
      ss_PackageID { ExternalAccessible := 'False'; ExternalVisible := 'False'; ExternalWritable := 'False'} : String[15];   // Identifier of Low-Level controls
      ss_Gap { ExternalAccessible := 'False'; ExternalVisible := 'False'; ExternalWritable := 'False'} : String[3];   // Gap converted to string
      sui_MsgArrayElNr { ExternalAccessible := 'False'; ExternalVisible := 'False'; ExternalWritable := 'False'} : UInt;   // Invalid message array size
      sui_ArrayOffset { ExternalAccessible := 'False'; ExternalVisible := 'False'; ExternalWritable := 'False'} : UInt;   // Offset for writing in the array
      si_OldGin { ExternalAccessible := 'False'; ExternalVisible := 'False'; ExternalWritable := 'False'} : Int;   // Previous Gin
      si_StringLen { ExternalAccessible := 'False'; ExternalVisible := 'False'; ExternalWritable := 'False'} : Int;   // Length of string used in loops to pad string with spaces or 0
      si_LenFillLoop { ExternalAccessible := 'False'; ExternalVisible := 'False'; ExternalWritable := 'False'} : Int;   // Loop couter
      si_MaxMsgLen { ExternalAccessible := 'False'; ExternalVisible := 'False'; ExternalWritable := 'False'} : Int;   // Maximum message length
      si_MsgLen { ExternalAccessible := 'False'; ExternalVisible := 'False'; ExternalWritable := 'False'} : Int;   // String character message length
      sx_Error { ExternalAccessible := 'False'; ExternalVisible := 'False'; ExternalWritable := 'False'} : Bool;
   END_VAR

   VAR CONSTANT
      cc_NULL : Char := '$00';   // NULL sign
      cc_STX : Char := '$02';   // Start of the text
      cc_ETX : Char := '$03';   // End of the text
      cs_Length : String := '0275';   // Legth of the message
      cs_MessageType : String := 'DX';   // Message type
   END_VAR


BEGIN
	(*
	----------------------------------------------------------------------------------------

	Version history:
	Date        | Version   | Author        | Remark
	----------------------------------------------------------------------------------------
	29/06/2021  | 1.0       | F.Baten       | first release MHS TIA 16.0
	10/11/2021  | 1.2       | M.Piela       | Updating regions numbering
	05/04/2022  | 1.3       | K.Pokorski    | Review
	21/02/2023  | 4.0       | F.Baten       | 4.0 Release TIA 17.5
	*)

	REGION 1 – FIFO header status update

	    // Mode 'S' - FIFO register status update
	    "FC_Fifo"(ic_Mode := 'S',
	              qUDT_Status => #sa_Status.FIFOStatus,
	              qx_Error => #sa_Status.FIFOError,
	              qx_Warning => #sa_Status.FIFOWarning,
	              iqv_Data := #sUDT_MessageArray,
	              iqUDT_FifoHeader := #iqUDT_FifoHeader,
	              iqv_DataBuffer := #iqa_FifoData);
	END_REGION

	REGION 2 - GIN validation

	    // GIN validation
	    #sa_Status.InvalidGIN :=
	    #ii_Gin < 1
	    OR #ii_Gin > 9999;

	END_REGION

	REGION 3 – Message preparation

	    IF NOT #iqUDT_FifoHeader.Status.Full       // FIFO isn't full
	        AND NOT #sa_Status.InvalidGIN
	        AND #ii_Gin <> #si_OldGin
	    THEN
	        REGION 3.1 - Sequencial ID
	            // ss_SequencialID character string clearing
	            #ss_SequencialID := '';
	            // ss_SequencialID integer input conversion to a character string
	            VAL_STRG(IN := "DB_GIN".GIN[#ii_Gin].FedEx.CustomerID,
	                     SIZE := 0,
	                     PREC := 0,
	                     FORMAT := 0,
	                     P := 1,
	                     OUT => #ss_SequencialID);
	            // Length of the ss_SequencialID character string
	            #si_StringLen := LEN(#ss_SequencialID);

